PROGRAM MAIN
VAR

	bInitial	:BOOL:= TRUE;;				//初始化
	ResetTrigger,AutoRunInitTrigger,PB_StartTrigger,IntiStartTrigger 	:R_TRIG;
	AutoRunDownTrigger,InitailDownTrigger	:F_TRIG;
	i	:INT;
END_VAR

//常態掃描  
RunParameter.strName	:= F_TrimRightSpace(RunParameter.strName);
Manual_POU();
IF PB_Stop OR PB_EMG OR OP.bStop_Sign THEN
	OP.xAutoRuning				:= FALSE;
	OP.xInitialRuning			:=FALSE;	
	OP.bInitialSign				:=FALSE;
	OP.xAutoMode				:=FALSE;
	RB_CS_SysIO.qENABLE			:= FALSE;
	RB_KR_SysIO.qMOVE_ENABLE	:= FALSE;
	
	MainControl.StopAllAxes();	
	MainControl.StopMotor();
	MainControl.StopAir();
END_IF
IF OP.bReset THEN
	MainControl.ErrorReset();
END_IF

(*---------------模式切換-------------------*)
IF OP.xAutoRuning OR OP.xAutoRuning THEN
	OP.bChangeMode	:=FALSE;
END_IF

IF OP.bChangeMode THEN
	OP.bChangeMode	:=FALSE;

	IF NOT OP.xAutoMode THEN
		EventLogger.eEventType	:= 1;
		EventLogger.strEventText	:= 'Mode : Auto ';
		EventLogger();
		OP.xAutoMode	:= TRUE;
		ELSE
		EventLogger.eEventType	:= 1;
		EventLogger.strEventText	:= 'Mode : Manual ';
		EventLogger();	
		OP.xAutoMode	:= FALSE;
	END_IF;
END_IF;
(*Stop*)



(*-------------POU Call ---------------*)
IF OP.xAutoRuning THEN
	OP.bInitialSign		:=FALSE;
END_IF;
IF NOT OP.xAutoMode THEN
	OP.xInitialDone	:=FALSE;
	OP.bStart		:=FALSE;
END_IF


PB_StartTrigger(CLK:=OP.bStart );
IntiStartTrigger(CLK:=OP.bInitialSign);
InitailDownTrigger(CLK:=OP.xInitialRuning);

IF OP.xAutoMode THEN
	IF IntiStartTrigger.Q THEN
		Initial_POU.FB_init(FALSE,FALSE);
		IF NOT OP.xAutoRuning THEN
			OP.xInitialRuning		:= TRUE;
			EventLogger.eEventType	:= 2;
			EventLogger.strEventText	:= 'Initial Runing ';
			EventLogger();
			ELSE
			EventLogger.eEventType	:= 4;
			EventLogger.strEventText	:= 'AutoRuning Do not Initial ';
			EventLogger();
		END_IF;
	END_IF;		
	IF PB_StartTrigger.Q AND NOT OP.xAutoRuning THEN
		IF NOT OP.xInitialRuning THEN
			OP.xAutoRuning	:= TRUE;
			EventLogger.eEventType	:= 2;
			EventLogger.strEventText	:= 'Auto Runing ';
			EventLogger();
			ELSE
			EventLogger.eEventType	:= 4;
			EventLogger.strEventText	:= 'Initial Runing,Please Waitting ';
			EventLogger();
		END_IF
	END_IF
END_IF

IF OP.xInitialRuning THEN
	Initial_POU();
END_IF
IF InitailDownTrigger.Q THEN
	MainControl.SoftStopAxis();
END_IF

IF OP.xAutoRuning THEN
	Automatic_POU();
END_IF

END_PROGRAM

(* stored: Version 1.1.0.1, ProductVersion 3.1.4024.16
   POU MAIN: Id {bbb2616a-be8a-4b16-b012-4fc48c768fe4}, SpecialFunc None *)
